// TIA Portal project "ozel_sayici" (V18)

(* hardware
DEVICE "S7-1200 station_1"  S7-1200 Station
   slot 0: "Rack_0"  S7-1200 Rack  Rack  V1.0
   slot 1: "PLC_1"  CPU 1214C DC/DC/DC  6ES7 214-1AG40-0XB0  V4.6
*)

// ===== PLC "PLC_1"  CPU 1214C DC/DC/DC =====

VAR_GLOBAL   // PLC tag table "Default tag table"
   "Tag_1" AT %I0.0 : Bool;
   "Tag_2" AT %I0.1 : Bool;
   "Tag_3" AT %I0.2 : Bool;
   "Tag_4" AT %MD0 : DInt;
   "Tag_5" AT %Q0.0 : Bool;
   "Tag_6" AT %Q0.1 : Bool;
END_VAR

DATA_BLOCK "Özel Sayıcı_DB"   // DB1
{ S7_Optimized_Access := 'TRUE' }
VERSION : 0.1
// stored: InstanceOfName Özel Sayıcı
"Özel Sayıcı"
BEGIN
END_DATA_BLOCK

FUNCTION_BLOCK "Özel Sayıcı"   // FB1, LAD
{ S7_Optimized_Access := 'TRUE' }
VERSION : 0.1
   VAR_INPUT
      ARTTIR : Bool;
      AZALT : Bool;
      ARTMA_MİKTARI : DInt;
      AZALMA_MİKTARI : DInt;
      ÜST_SINIR : DInt;
      ALT_SINIR : DInt;
      SİLME : Bool;
   END_VAR
   VAR_OUTPUT
      ÜST_ÇIKIŞ : Bool;
      ALT_ÇIKIŞ : Bool;
   END_VAR
   VAR_IN_OUT
      SAYICI_İÇERİĞİ : DInt;
   END_VAR
   VAR
      "ARTIŞ DARBE" : Bool;
      "AZALIŞ DARBE" : Bool;
   END_VAR
   VAR_TEMP   // added for the SCL form of the ladder/FBD networks
      _w1 : Bool;
   END_VAR
BEGIN

REGION Network 1
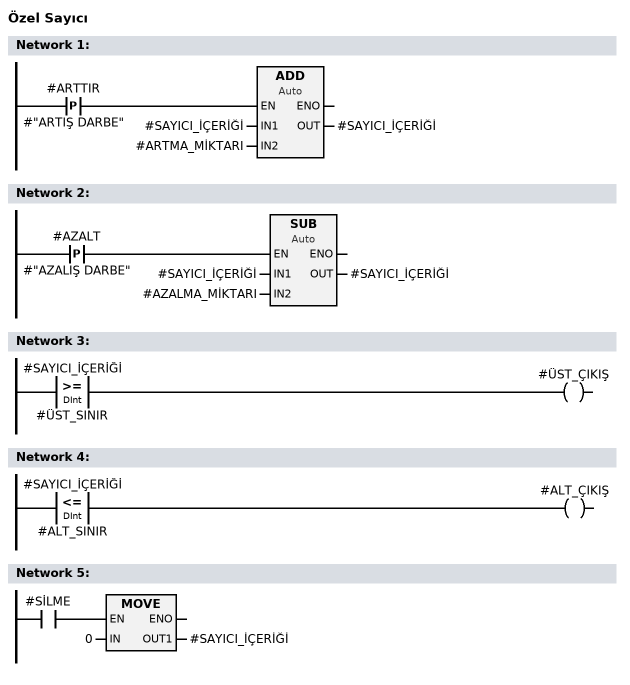
   RUNG wire#powerrail
      P_Contact(operand := #ARTTIR, bit := #"ARTIŞ DARBE")
      Add(in1 := #SAYICI_İÇERİĞİ, in2 := #ARTMA_MİKTARI, out => #SAYICI_İÇERİĞİ)
   END_RUNG
   // the same network as SCL:
   #_w1 := #ARTTIR AND NOT #"ARTIŞ DARBE";   // rising edge of #ARTTIR
   #"ARTIŞ DARBE" := #ARTTIR;
   IF #_w1 THEN #SAYICI_İÇERİĞİ := #SAYICI_İÇERİĞİ + #ARTMA_MİKTARI; END_IF;
END_REGION

REGION Network 2
   RUNG wire#powerrail
      P_Contact(operand := #AZALT, bit := #"AZALIŞ DARBE")
      Sub(in1 := #SAYICI_İÇERİĞİ, in2 := #AZALMA_MİKTARI, out => #SAYICI_İÇERİĞİ)
   END_RUNG
   // the same network as SCL:
   #_w1 := #AZALT AND NOT #"AZALIŞ DARBE";   // rising edge of #AZALT
   #"AZALIŞ DARBE" := #AZALT;
   IF #_w1 THEN #SAYICI_İÇERİĞİ := #SAYICI_İÇERİĞİ - #AZALMA_MİKTARI; END_IF;
END_REGION

REGION Network 3
   RUNG wire#powerrail
      { S7_Templates := "SrcType := DInt" } GE_Contact(in1 := #SAYICI_İÇERİĞİ, in2 := #ÜST_SINIR)
      Coil( #ÜST_ÇIKIŞ )
   END_RUNG
   // the same network as SCL:
   #ÜST_ÇIKIŞ := #SAYICI_İÇERİĞİ >= #ÜST_SINIR;
END_REGION

REGION Network 4
   RUNG wire#powerrail
      { S7_Templates := "SrcType := DInt" } LE_Contact(in1 := #SAYICI_İÇERİĞİ, in2 := #ALT_SINIR)
      Coil( #ALT_ÇIKIŞ )
   END_RUNG
   // the same network as SCL:
   #ALT_ÇIKIŞ := #SAYICI_İÇERİĞİ <= #ALT_SINIR;
END_REGION

REGION Network 5
   RUNG wire#powerrail
      Contact( #SİLME )
      Move(in := 0, out1 => #SAYICI_İÇERİĞİ)
   END_RUNG
   // the same network as SCL:
   IF #SİLME THEN #SAYICI_İÇERİĞİ := 0; END_IF;
END_REGION
END_FUNCTION_BLOCK

ORGANIZATION_BLOCK "Main"   // OB1, LAD, ProgramCycle
TITLE = "Main Program Sweep (Cycle)"
{ S7_Optimized_Access := 'TRUE' }
VERSION : 0.1
   VAR_INPUT
      Initial_Call : Bool;   // Initial call of this OB
      Remanence : Bool;   // =True, if remanent data are available
   END_VAR
BEGIN

REGION Network 1
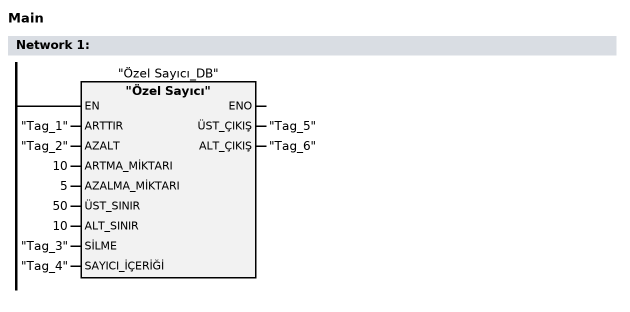
   RUNG wire#powerrail
      "Özel Sayıcı_DB"(ARTTIR := "Tag_1", AZALT := "Tag_2", ARTMA_MİKTARI := 10, AZALMA_MİKTARI := 5, ÜST_SINIR := 50, ALT_SINIR := 10, SİLME := "Tag_3", SAYICI_İÇERİĞİ := "Tag_4", ÜST_ÇIKIŞ => "Tag_5", ALT_ÇIKIŞ => "Tag_6")
   END_RUNG
   // the same network as SCL:
   "Özel Sayıcı_DB"(ARTTIR := "Tag_1",   // "Özel Sayıcı"
                    AZALT := "Tag_2",
                    ARTMA_MİKTARI := 10,
                    AZALMA_MİKTARI := 5,
                    ÜST_SINIR := 50,
                    ALT_SINIR := 10,
                    SİLME := "Tag_3",
                    SAYICI_İÇERİĞİ := "Tag_4",
                    ÜST_ÇIKIŞ => "Tag_5",
                    ALT_ÇIKIŞ => "Tag_6");
END_REGION
END_ORGANIZATION_BLOCK